PROGRAM FB_Motion1way
VAR
END_VAR

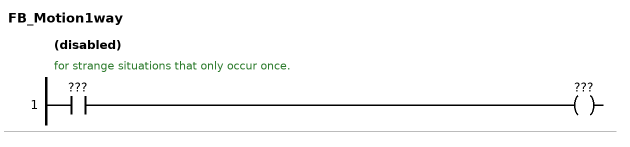
// NETWORK 1 (disabled)
// for strange situations that only occur once.
// ??? := ???;

END_PROGRAM

(* stored: Version 1.1.0.1, ProductVersion 3.1.4024.12
   POU FB_Motion1way: Id {94bc97ff-8896-4204-82e1-db7f8bcefc22}, SpecialFunc None *)
